FUNCTION_BLOCK FB_GetStateAutoRow
VAR_INPUT
	iRowNumber:UINT; //the row number for the motion

	iIsAdvanced:BOOL; //TRUE if the motion is advanced (depth)
	iIsReturned:BOOL; //TRUE if the motion is returned (depth)
	
	//iNextStepNum:UINT; //should just be +1
END_VAR
VAR_OUTPUT
	qPerformAdvance:BOOL; //TRUE to get the motion block to perform the motion (advance)
	qPerformReturn:BOOL; //TRUE to get the motion block to perform the motion (return)
END_VAR
VAR
	tStepIsLastStep: BOOL;
END_VAR
VAR_IN_OUT
	stndata:typeStation;
	SeqData:typeRowHolder;
END_VAR
VAR // added by the converter: edge detectors and wires of the graphical bodies
    _rt1, _rt2 : R_TRIG;
END_VAR

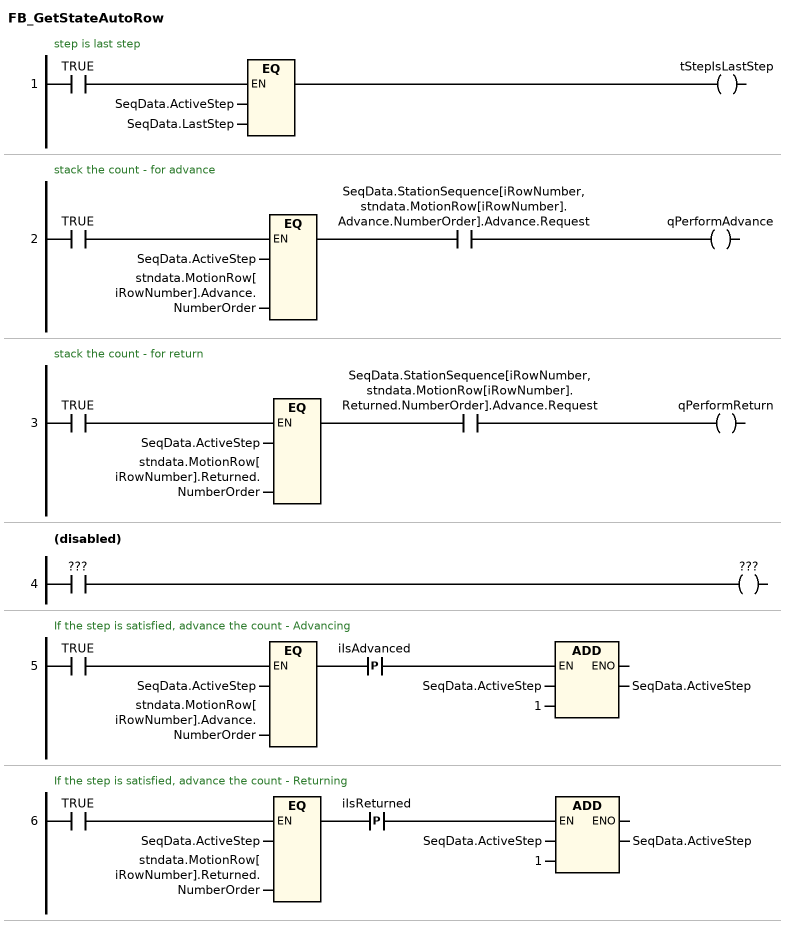
// NETWORK 1
// step is last step
tStepIsLastStep := SeqData.ActiveStep = SeqData.LastStep;

// NETWORK 2
// stack the count - for advance
qPerformAdvance := SeqData.ActiveStep = stndata.MotionRow[iRowNumber].Advance.NumberOrder AND (SeqData.StationSequence[iRowNumber,stndata.MotionRow[iRowNumber].Advance.NumberOrder].Advance.Request);

// NETWORK 3
// stack the count - for return
qPerformReturn := SeqData.ActiveStep = stndata.MotionRow[iRowNumber].Returned.NumberOrder AND (SeqData.StationSequence[iRowNumber,stndata.MotionRow[iRowNumber].Returned.NumberOrder].Advance.Request);

// NETWORK 4 (disabled)
// ??? := ???;

// NETWORK 5
// If the step is satisfied, advance the count - Advancing
_rt1(CLK := iIsAdvanced);
IF SeqData.ActiveStep = stndata.MotionRow[iRowNumber].Advance.NumberOrder AND _rt1.Q THEN
    SeqData.ActiveStep := SeqData.ActiveStep + 1;
END_IF

// NETWORK 6
// If the step is satisfied, advance the count - Returning
_rt2(CLK := iIsReturned);
IF SeqData.ActiveStep = stndata.MotionRow[iRowNumber].Returned.NumberOrder AND _rt2.Q THEN
    SeqData.ActiveStep := SeqData.ActiveStep + 1;
END_IF

END_FUNCTION_BLOCK

(* stored: Version 1.1.0.1, ProductVersion 3.1.4024.11
   POU FB_GetStateAutoRow: Id {50eadc3e-ccea-07c0-04c6-2cabdc9f5d2e}, SpecialFunc None *)
